{attribute 'pack_mode' := '2'}
TYPE ST_XPU_CTRL :
STRUCT
  Cmd             : E_XPU_CTRL;
END_STRUCT
END_TYPE

(* stored: Version 1.1.0.1
   DUT ST_XPU_CTRL: Id {4d81e152-e021-4acc-a2de-772e9d8c9d55} *)
